Staubli VAL3: onF2Event.pgx

program onF2Event()
  local string l_sEmpty
begin
  // look if the bButton is enable
  if bButton[1]
    // tool selection
    call loadPage("Disk://kernel/page/tool",l_sEmpty)
    //
    saveData:nFrameTool=saveData:nIndexTool
  endIf
end
